PROGRAM AuxiliaryControl
VAR
	// start delay for the dehumidifier to prevent overcurrent
	pressure_voltage,
	pressure_Dewar,
	temperature_Dewar: REAL;
END_VAR

// turn off dehumidifier if dome is open
pressure_voltage := F_YREAL(GVL_Auxiliary.pressure_Dewar, 0, 32767, 0.0, 10.0);
pressure_Dewar := LREAL_TO_REAL(EXPT(10.0, (1.5*pressure_voltage - 12.0)));
temperature_Dewar := GVL_Auxiliary.temperature_Dewar / 100.0;

END_PROGRAM

(* stored: Version 1.1.0.1, ProductVersion 3.1.4024.9
   POU AuxiliaryControl: Id {30a3eb2e-ebab-4f9f-a38d-cee5e71b2e38}, SpecialFunc None *)
